(* IEC 61131-3 sources: Wago_IOWalkTest/Device/Application/FBs, 4 files *)

(* ---- FB_AITest.st ---- *)
FUNCTION_BLOCK FB_AITest
VAR_INPUT
    bStart          : BOOL;
    bStop           : BOOL;
    bSkip           : BOOL;
    bContinue       : BOOL;        // Operator presses between passes
    bStartWireBreak : BOOL;        // Start optional wire break pass
    bRetestOnly     : BOOL;
END_VAR
VAR_OUTPUT
    eState          : E_TestState;
    nCurrentChannel : INT;
    nCurrentPass    : INT;         // 1=4mA, 2=12mA, 3=20mA, 4=wirebreak
    nTotalChannels  : INT := GVL_IOWalkTest.C_NUM_AI;
    aReadings       : ARRAY[0..31, 1..3] OF INT;
    aResults        : ARRAY[0..31, 1..4] OF E_TestResult;  // 4th = wire break
    sCurrentAddress : STRING(15);
    sCurrentTag     : STRING(40);
    sCurrentDesc    : STRING(80);
    sCurrentUnit    : STRING(15);
    nCurrentRaw     : INT;
    nExpectedRaw    : INT;
    rCurrentScaled  : REAL;
    rExpectedScaled : REAL;
    rErrorPct       : REAL;
    rMaxErrorPct    : REAL;
    bSignalDetected : BOOL;
    bSettling       : BOOL;
    nPassed         : INT;
    nFailed         : INT;
    bAlmTimeout     : BOOL;
    bWireBreakDone  : BOOL;
END_VAR
VAR
    fbSettle        : TON;
    fbTimeout       : TON;
    aAI_Channels    : ARRAY[0..31] OF ST_AIChannel;
    bStartPrev      : BOOL;
    bSkipPrev       : BOOL;
    bContinuePrev   : BOOL;
    bWireBreakPrev  : BOOL;
    i               : INT;
    nRaw            : INT;
    bInWindow       : BOOL;
    rScaledActual   : REAL;
    rScaledExpected : REAL;
    rSpan           : REAL;
    rErr            : REAL;
END_VAR

// One-shot start
IF bStart AND NOT bStartPrev THEN
    IF eState = E_TestState.IDLE OR eState = E_TestState.COMPLETE OR eState = E_TestState.ABORTED THEN
        eState := E_TestState.RUNNING;
        nCurrentChannel := 0;
        nCurrentPass := 1;
        nPassed := 0;
        nFailed := 0;
        rMaxErrorPct := 0.0;
        bAlmTimeout := FALSE;
        bWireBreakDone := FALSE;
        fbSettle(IN := FALSE);
        fbTimeout(IN := FALSE);

        IF NOT bRetestOnly THEN
            FOR i := 0 TO 31 DO
                aResults[i, 1] := E_TestResult.UNTESTED;
                aResults[i, 2] := E_TestResult.UNTESTED;
                aResults[i, 3] := E_TestResult.UNTESTED;
                aResults[i, 4] := E_TestResult.UNTESTED;
            END_FOR
        END_IF
    END_IF
END_IF
bStartPrev := bStart;

// Stop
IF bStop THEN
    IF eState = E_TestState.RUNNING OR eState = E_TestState.WAIT_CONTINUE THEN
        eState := E_TestState.ABORTED;
        fbSettle(IN := FALSE);
        fbTimeout(IN := FALSE);
    END_IF
END_IF

// Continue between passes (one-shot)
IF bContinue AND NOT bContinuePrev AND eState = E_TestState.WAIT_CONTINUE THEN
    eState := E_TestState.RUNNING;
    fbTimeout(IN := FALSE);
END_IF
bContinuePrev := bContinue;

// Skip channel (one-shot)
IF bSkip AND NOT bSkipPrev AND eState = E_TestState.RUNNING THEN
    aResults[nCurrentChannel, nCurrentPass] := E_TestResult.SKIPPED;
    fbSettle(IN := FALSE);
    fbTimeout(IN := FALSE);
    nCurrentChannel := nCurrentChannel + 1;

    IF nCurrentChannel >= nTotalChannels THEN
        IF nCurrentPass < 3 THEN
            eState := E_TestState.WAIT_CONTINUE;
            nCurrentChannel := 0;
            nCurrentPass := nCurrentPass + 1;
        ELSE
            eState := E_TestState.COMPLETE;
        END_IF
    END_IF
END_IF
bSkipPrev := bSkip;

// Wire break test (one-shot)
IF bStartWireBreak AND NOT bWireBreakPrev THEN
    IF eState = E_TestState.COMPLETE OR eState = E_TestState.IDLE THEN
        nCurrentPass := 4;
        bWireBreakDone := FALSE;

        FOR i := 0 TO nTotalChannels - 1 DO
            IF aAI_Channels[i].pInput <> 0 THEN
                nRaw := aAI_Channels[i].pInput^;
                IF nRaw < GVL_IOWalkTest.C_AI_WIREBREAK_MAX THEN
                    aResults[i, 4] := E_TestResult.PASSED;
                    nPassed := nPassed + 1;
                ELSE
                    aResults[i, 4] := E_TestResult.FAILED;
                    nFailed := nFailed + 1;
                END_IF
            END_IF
        END_FOR

        bWireBreakDone := TRUE;
    END_IF
END_IF
bWireBreakPrev := bStartWireBreak;

// Main test logic (passes 1-3)
IF eState = E_TestState.RUNNING AND nCurrentPass >= 1 AND nCurrentPass <= 3
   AND nCurrentChannel < nTotalChannels THEN

    // Update HMI info
    sCurrentAddress := aAI_Channels[nCurrentChannel].sAddress;
    sCurrentTag     := aAI_Channels[nCurrentChannel].sTag;
    sCurrentDesc    := aAI_Channels[nCurrentChannel].sDescription;
    sCurrentUnit    := aAI_Channels[nCurrentChannel].sUnit;
    nExpectedRaw    := GVL_IOWalkTest.C_AI_EXPECTED_RAW[nCurrentPass];

    // Read current raw value
    IF aAI_Channels[nCurrentChannel].pInput <> 0 THEN
        nCurrentRaw := aAI_Channels[nCurrentChannel].pInput^;
    END_IF

    // Scale for display
    rSpan := aAI_Channels[nCurrentChannel].rRangeHigh - aAI_Channels[nCurrentChannel].rRangeLow;
    IF rSpan > 0.0 THEN
        rCurrentScaled  := aAI_Channels[nCurrentChannel].rRangeLow
                           + (INT_TO_REAL(nCurrentRaw) / 32767.0) * rSpan;
        rExpectedScaled := aAI_Channels[nCurrentChannel].rRangeLow
                           + (INT_TO_REAL(nExpectedRaw) / 32767.0) * rSpan;
    END_IF

    // Channel timeout
    fbTimeout(IN := TRUE, PT := GVL_IOWalkTest.C_AI_TIMEOUT);

    // Check if signal is within expected window
    bInWindow := ABS(nCurrentRaw - nExpectedRaw) < GVL_IOWalkTest.C_AI_RAW_TOLERANCE;
    bSignalDetected := bInWindow;

    IF bInWindow THEN
        // Settle timer
        fbSettle(IN := TRUE, PT := GVL_IOWalkTest.C_AI_SETTLE_TIME);
        bSettling := TRUE;

        IF fbSettle.Q THEN
            // Record reading
            aReadings[nCurrentChannel, nCurrentPass] := nCurrentRaw;

            // Evaluate pass/fail
            rScaledActual   := aAI_Channels[nCurrentChannel].rRangeLow
                               + (INT_TO_REAL(nCurrentRaw) / 32767.0) * rSpan;
            rScaledExpected := aAI_Channels[nCurrentChannel].rRangeLow
                               + (INT_TO_REAL(nExpectedRaw) / 32767.0) * rSpan;

            IF rSpan > 0.0 THEN
                rErr := ABS(rScaledActual - rScaledExpected) / rSpan * 100.0;
            ELSE
                rErr := 0.0;
            END_IF

            rErrorPct := rErr;
            IF rErr > rMaxErrorPct THEN
                rMaxErrorPct := rErr;
            END_IF

            IF rErr < GVL_IOWalkTest.C_AI_ERROR_PCT_MAX THEN
                aResults[nCurrentChannel, nCurrentPass] := E_TestResult.PASSED;
                nPassed := nPassed + 1;
            ELSE
                aResults[nCurrentChannel, nCurrentPass] := E_TestResult.FAILED;
                nFailed := nFailed + 1;
            END_IF

            // Advance
            fbSettle(IN := FALSE);
            fbTimeout(IN := FALSE);
            bSettling := FALSE;
            nCurrentChannel := nCurrentChannel + 1;

            IF nCurrentChannel >= nTotalChannels THEN
                IF nCurrentPass < 3 THEN
                    eState := E_TestState.WAIT_CONTINUE;
                    nCurrentChannel := 0;
                    nCurrentPass := nCurrentPass + 1;
                ELSE
                    eState := E_TestState.COMPLETE;
                END_IF
            END_IF
        END_IF
    ELSE
        fbSettle(IN := FALSE);
        bSettling := FALSE;
    END_IF

    // Timeout
    IF fbTimeout.Q THEN
        aResults[nCurrentChannel, nCurrentPass] := E_TestResult.FAILED;
        nFailed := nFailed + 1;
        bAlmTimeout := TRUE;
        fbSettle(IN := FALSE);
        fbTimeout(IN := FALSE);
        bSettling := FALSE;
        nCurrentChannel := nCurrentChannel + 1;

        IF nCurrentChannel >= nTotalChannels THEN
            IF nCurrentPass < 3 THEN
                eState := E_TestState.WAIT_CONTINUE;
                nCurrentChannel := 0;
                nCurrentPass := nCurrentPass + 1;
            ELSE
                eState := E_TestState.COMPLETE;
            END_IF
        END_IF
    END_IF
END_IF

(* ---- FB_AOTest.st ---- *)
FUNCTION_BLOCK FB_AOTest
VAR_INPUT
    bStart      : BOOL;
    bStop       : BOOL;
    bSkip       : BOOL;
    bPause      : BOOL;
    bMarkFail   : BOOL;
    bRetestOnly : BOOL;
END_VAR
VAR_OUTPUT
    eState          : E_TestState;
    nCurrentChannel : INT;
    nTotalChannels  : INT := GVL_IOWalkTest.C_NUM_AO;
    aResults        : ARRAY[0..11] OF E_TestResult;
    ePhase          : E_AOPhase;
    sCurrentAddress : STRING(15);
    sCurrentTag     : STRING(40);
    sCurrentDesc    : STRING(80);
    sNextAddress    : STRING(15);
    sNextTag        : STRING(40);
    rCurrentOutput_mA : REAL;
    rRampProgress   : REAL;       // 0.0 to 1.0
    nPassed         : INT;
    nFailed         : INT;
    nSkipped        : INT;
END_VAR
VAR
    fbRampTimer     : TON;
    aAO_Channels    : ARRAY[0..11] OF ST_AOChannel;
    bStartPrev      : BOOL;
    bSkipPrev       : BOOL;
    bMarkFailPrev   : BOOL;
    bChannelMarkedFail : BOOL;
    nOutputRaw      : INT;
    rProgress       : REAL;
    tCurrentPT      : TIME;
    i               : INT;
END_VAR

// One-shot start
IF bStart AND NOT bStartPrev THEN
    IF eState = E_TestState.IDLE OR eState = E_TestState.COMPLETE OR eState = E_TestState.ABORTED THEN
        eState := E_TestState.RUNNING;
        nCurrentChannel := 0;
        ePhase := E_AOPhase.RAMP_UP;
        nPassed := 0;
        nFailed := 0;
        nSkipped := 0;
        bChannelMarkedFail := FALSE;
        fbRampTimer(IN := FALSE);

        IF NOT bRetestOnly THEN
            FOR i := 0 TO 11 DO
                aResults[i] := E_TestResult.UNTESTED;
            END_FOR
        END_IF

        // Zero all outputs
        FOR i := 0 TO 11 DO
            IF aAO_Channels[i].pOutput <> 0 THEN
                aAO_Channels[i].pOutput^ := 0;
            END_IF
        END_FOR

        IF bRetestOnly THEN
            WHILE nCurrentChannel < nTotalChannels
                  AND aResults[nCurrentChannel] = E_TestResult.PASSED DO
                nCurrentChannel := nCurrentChannel + 1;
            END_WHILE
        END_IF
    END_IF
END_IF
bStartPrev := bStart;

// Stop / All Off
IF bStop THEN
    FOR i := 0 TO 11 DO
        IF aAO_Channels[i].pOutput <> 0 THEN
            aAO_Channels[i].pOutput^ := 0;
        END_IF
    END_FOR
    IF eState = E_TestState.RUNNING OR eState = E_TestState.PAUSED THEN
        eState := E_TestState.ABORTED;
        fbRampTimer(IN := FALSE);
    END_IF
END_IF

// Pause toggle
IF bPause AND eState = E_TestState.RUNNING THEN
    eState := E_TestState.PAUSED;
ELSIF bPause AND eState = E_TestState.PAUSED THEN
    eState := E_TestState.RUNNING;
END_IF

// Skip (one-shot)
IF bSkip AND NOT bSkipPrev AND eState = E_TestState.RUNNING THEN
    IF aAO_Channels[nCurrentChannel].pOutput <> 0 THEN
        aAO_Channels[nCurrentChannel].pOutput^ := 0;
    END_IF
    aResults[nCurrentChannel] := E_TestResult.SKIPPED;
    nSkipped := nSkipped + 1;
    bChannelMarkedFail := FALSE;
    fbRampTimer(IN := FALSE);
    ePhase := E_AOPhase.RAMP_UP;
    nCurrentChannel := nCurrentChannel + 1;

    IF bRetestOnly THEN
        WHILE nCurrentChannel < nTotalChannels
              AND aResults[nCurrentChannel] = E_TestResult.PASSED DO
            nCurrentChannel := nCurrentChannel + 1;
        END_WHILE
    END_IF

    IF nCurrentChannel >= nTotalChannels THEN
        eState := E_TestState.COMPLETE;
    END_IF
END_IF
bSkipPrev := bSkip;

// Mark fail (one-shot)
IF bMarkFail AND NOT bMarkFailPrev AND eState = E_TestState.RUNNING THEN
    bChannelMarkedFail := TRUE;
END_IF
bMarkFailPrev := bMarkFail;

// Main ramp logic
IF eState = E_TestState.RUNNING AND nCurrentChannel < nTotalChannels THEN
    // HMI info
    sCurrentAddress := aAO_Channels[nCurrentChannel].sAddress;
    sCurrentTag     := aAO_Channels[nCurrentChannel].sTag;
    sCurrentDesc    := aAO_Channels[nCurrentChannel].sDescription;

    IF nCurrentChannel + 1 < nTotalChannels THEN
        sNextAddress := aAO_Channels[nCurrentChannel + 1].sAddress;
        sNextTag     := aAO_Channels[nCurrentChannel + 1].sTag;
    ELSE
        sNextAddress := '';
        sNextTag     := '(last channel)';
    END_IF

    // Select timer preset based on phase
    CASE ePhase OF
        E_AOPhase.RAMP_UP, E_AOPhase.RAMP_DOWN:
            tCurrentPT := GVL_IOWalkTest.C_AO_RAMP_TIME;
        E_AOPhase.PAUSE:
            tCurrentPT := GVL_IOWalkTest.C_AO_PAUSE_TIME;
    END_CASE

    fbRampTimer(IN := TRUE, PT := tCurrentPT);
    rProgress := TIME_TO_REAL(fbRampTimer.ET) / TIME_TO_REAL(tCurrentPT);
    IF rProgress > 1.0 THEN rProgress := 1.0; END_IF
    rRampProgress := rProgress;

    CASE ePhase OF
    E_AOPhase.RAMP_UP:
        // 4mA -> 20mA (raw 0 -> 32767)
        nOutputRaw := REAL_TO_INT(rProgress * 32767.0);
        IF aAO_Channels[nCurrentChannel].pOutput <> 0 THEN
            aAO_Channels[nCurrentChannel].pOutput^ := nOutputRaw;
        END_IF
        rCurrentOutput_mA := 4.0 + (rProgress * 16.0);

        IF fbRampTimer.Q THEN
            fbRampTimer(IN := FALSE);
            ePhase := E_AOPhase.RAMP_DOWN;
        END_IF

    E_AOPhase.RAMP_DOWN:
        // 20mA -> 4mA (raw 32767 -> 0)
        nOutputRaw := REAL_TO_INT((1.0 - rProgress) * 32767.0);
        IF aAO_Channels[nCurrentChannel].pOutput <> 0 THEN
            aAO_Channels[nCurrentChannel].pOutput^ := nOutputRaw;
        END_IF
        rCurrentOutput_mA := 4.0 + ((1.0 - rProgress) * 16.0);

        IF fbRampTimer.Q THEN
            IF aAO_Channels[nCurrentChannel].pOutput <> 0 THEN
                aAO_Channels[nCurrentChannel].pOutput^ := 0;
            END_IF
            fbRampTimer(IN := FALSE);
            ePhase := E_AOPhase.PAUSE;
        END_IF

    E_AOPhase.PAUSE:
        // Pause between channels
        IF aAO_Channels[nCurrentChannel].pOutput <> 0 THEN
            aAO_Channels[nCurrentChannel].pOutput^ := 0;
        END_IF
        rCurrentOutput_mA := 4.0;

        IF fbRampTimer.Q THEN
            // Record result
            IF bChannelMarkedFail THEN
                aResults[nCurrentChannel] := E_TestResult.FAILED;
                nFailed := nFailed + 1;
            ELSE
                aResults[nCurrentChannel] := E_TestResult.PASSED;
                nPassed := nPassed + 1;
            END_IF

            bChannelMarkedFail := FALSE;
            fbRampTimer(IN := FALSE);
            ePhase := E_AOPhase.RAMP_UP;
            nCurrentChannel := nCurrentChannel + 1;

            IF bRetestOnly THEN
                WHILE nCurrentChannel < nTotalChannels
                      AND aResults[nCurrentChannel] = E_TestResult.PASSED DO
                    nCurrentChannel := nCurrentChannel + 1;
                END_WHILE
            END_IF

            IF nCurrentChannel >= nTotalChannels THEN
                FOR i := 0 TO 11 DO
                    IF aAO_Channels[i].pOutput <> 0 THEN
                        aAO_Channels[i].pOutput^ := 0;
                    END_IF
                END_FOR
                eState := E_TestState.COMPLETE;
            END_IF
        END_IF
    END_CASE
END_IF

(* ---- FB_DITest.st ---- *)
FUNCTION_BLOCK FB_DITest
VAR_INPUT
    bStart          : BOOL;
    bStop           : BOOL;
    bSkip           : BOOL;
    bRetestOnly     : BOOL;     // Only retest channels that previously failed
END_VAR
VAR_OUTPUT
    eState          : E_TestState;
    nCurrentChannel : INT;
    nTotalChannels  : INT := GVL_IOWalkTest.C_NUM_DI;
    aResults        : ARRAY[0..71] OF E_TestResult;
    bWaitingForRise : BOOL;
    bWaitingForFall : BOOL;
    sCurrentAddress : STRING(15);
    sCurrentTag     : STRING(40);
    sCurrentDesc    : STRING(80);
    eCurrentContact : E_ContactType;
    nPassed         : INT;
    nFailed         : INT;
    nSkipped        : INT;
    bAlmTimeout     : BOOL;
    bAlmWrongChan   : BOOL;
    nWrongChanIdx   : INT;
END_VAR
VAR
    fbTimeout       : TON;
    aDI_Prev        : ARRAY[0..71] OF BOOL;
    aDI_Channels    : ARRAY[0..71] OF ST_DIChannel;
    bInitDone       : BOOL;
    bStartPrev      : BOOL;
    bSkipPrev       : BOOL;
    i               : INT;
    bCurrentState   : BOOL;
    bPrevState      : BOOL;
    bExpectRise     : BOOL;     // TRUE = waiting for active edge
    bExpectFall     : BOOL;     // TRUE = waiting for release edge
END_VAR

// One-shot start detection
IF bStart AND NOT bStartPrev THEN
    IF eState = E_TestState.IDLE OR eState = E_TestState.COMPLETE OR eState = E_TestState.ABORTED THEN
        eState := E_TestState.RUNNING;
        nCurrentChannel := 0;
        bAlmTimeout := FALSE;
        bAlmWrongChan := FALSE;
        nPassed := 0;
        nFailed := 0;
        nSkipped := 0;
        fbTimeout(IN := FALSE);

        IF NOT bRetestOnly THEN
            FOR i := 0 TO 71 DO
                aResults[i] := E_TestResult.UNTESTED;
            END_FOR
        END_IF

        // Skip to first untested/failed channel if retest mode
        IF bRetestOnly THEN
            WHILE nCurrentChannel < nTotalChannels
                  AND aResults[nCurrentChannel] = E_TestResult.PASSED DO
                nCurrentChannel := nCurrentChannel + 1;
            END_WHILE
        END_IF

        // Determine initial edge expectations
        IF nCurrentChannel < nTotalChannels THEN
            IF aDI_Channels[nCurrentChannel].eContactType = E_ContactType.NC THEN
                bExpectRise := FALSE;
                bExpectFall := TRUE;    // NC: wait for fall first
            ELSE
                bExpectRise := TRUE;
                bExpectFall := FALSE;   // NO: wait for rise first
            END_IF
        END_IF
    END_IF
END_IF
bStartPrev := bStart;

// Stop
IF bStop THEN
    IF eState = E_TestState.RUNNING THEN
        eState := E_TestState.ABORTED;
        fbTimeout(IN := FALSE);
    END_IF
END_IF

// Skip channel (one-shot)
IF bSkip AND NOT bSkipPrev AND eState = E_TestState.RUNNING THEN
    aResults[nCurrentChannel] := E_TestResult.SKIPPED;
    nSkipped := nSkipped + 1;
    fbTimeout(IN := FALSE);
    nCurrentChannel := nCurrentChannel + 1;

    // Skip already-passed channels in retest mode
    IF bRetestOnly THEN
        WHILE nCurrentChannel < nTotalChannels
              AND aResults[nCurrentChannel] = E_TestResult.PASSED DO
            nCurrentChannel := nCurrentChannel + 1;
        END_WHILE
    END_IF

    IF nCurrentChannel >= nTotalChannels THEN
        eState := E_TestState.COMPLETE;
    END_IF
END_IF
bSkipPrev := bSkip;

// Main test logic
IF eState = E_TestState.RUNNING AND nCurrentChannel < nTotalChannels THEN
    // Update HMI display info
    sCurrentAddress := aDI_Channels[nCurrentChannel].sAddress;
    sCurrentTag     := aDI_Channels[nCurrentChannel].sTag;
    sCurrentDesc    := aDI_Channels[nCurrentChannel].sDescription;
    eCurrentContact := aDI_Channels[nCurrentChannel].eContactType;

    // Read current channel state via pointer
    IF aDI_Channels[nCurrentChannel].pInput <> 0 THEN
        bCurrentState := aDI_Channels[nCurrentChannel].pInput^;
    END_IF
    bPrevState := aDI_Prev[nCurrentChannel];

    // Channel timeout
    fbTimeout(IN := TRUE, PT := GVL_IOWalkTest.C_DI_TIMEOUT);

    // Edge detection based on contact type
    // NO contacts: rise then fall
    // NC contacts: fall then rise (inverted)
    IF bExpectRise AND bCurrentState AND NOT bPrevState THEN
        // Rising edge detected
        bExpectRise := FALSE;
        bExpectFall := TRUE;
        fbTimeout(IN := FALSE);
        fbTimeout(IN := TRUE, PT := GVL_IOWalkTest.C_DI_TIMEOUT);
    END_IF

    IF bExpectFall AND NOT bCurrentState AND bPrevState THEN
        // Falling edge detected - channel PASS
        aResults[nCurrentChannel] := E_TestResult.PASSED;
        nPassed := nPassed + 1;
        fbTimeout(IN := FALSE);

        // Advance
        nCurrentChannel := nCurrentChannel + 1;

        // Skip already-passed in retest mode
        IF bRetestOnly THEN
            WHILE nCurrentChannel < nTotalChannels
                  AND aResults[nCurrentChannel] = E_TestResult.PASSED DO
                nCurrentChannel := nCurrentChannel + 1;
            END_WHILE
        END_IF

        IF nCurrentChannel >= nTotalChannels THEN
            eState := E_TestState.COMPLETE;
        ELSE
            // Set up edge expectations for next channel
            IF aDI_Channels[nCurrentChannel].eContactType = E_ContactType.NC THEN
                bExpectRise := FALSE;
                bExpectFall := TRUE;
            ELSE
                bExpectRise := TRUE;
                bExpectFall := FALSE;
            END_IF
            fbTimeout(IN := TRUE, PT := GVL_IOWalkTest.C_DI_TIMEOUT);
        END_IF
    END_IF

    // Check for out-of-order channel activation
    FOR i := 0 TO nTotalChannels - 1 DO
        IF i <> nCurrentChannel AND aDI_Channels[i].pInput <> 0 THEN
            IF aDI_Channels[i].pInput^ AND NOT aDI_Prev[i] THEN
                bAlmWrongChan := TRUE;
                nWrongChanIdx := i;
            END_IF
        END_IF
    END_FOR

    // Timeout handling
    IF fbTimeout.Q THEN
        aResults[nCurrentChannel] := E_TestResult.FAILED;
        nFailed := nFailed + 1;
        bAlmTimeout := TRUE;
        fbTimeout(IN := FALSE);

        nCurrentChannel := nCurrentChannel + 1;
        IF bRetestOnly THEN
            WHILE nCurrentChannel < nTotalChannels
                  AND aResults[nCurrentChannel] = E_TestResult.PASSED DO
                nCurrentChannel := nCurrentChannel + 1;
            END_WHILE
        END_IF

        IF nCurrentChannel >= nTotalChannels THEN
            eState := E_TestState.COMPLETE;
        ELSE
            IF aDI_Channels[nCurrentChannel].eContactType = E_ContactType.NC THEN
                bExpectRise := FALSE;
                bExpectFall := TRUE;
            ELSE
                bExpectRise := TRUE;
                bExpectFall := FALSE;
            END_IF
            fbTimeout(IN := TRUE, PT := GVL_IOWalkTest.C_DI_TIMEOUT);
        END_IF
    END_IF

    // Store previous states for all channels
    FOR i := 0 TO nTotalChannels - 1 DO
        IF aDI_Channels[i].pInput <> 0 THEN
            aDI_Prev[i] := aDI_Channels[i].pInput^;
        END_IF
    END_FOR
END_IF

(* ---- FB_DOTest.st ---- *)
FUNCTION_BLOCK FB_DOTest
VAR_INPUT
    bStart      : BOOL;
    bStop       : BOOL;
    bSkip       : BOOL;
    bPause      : BOOL;
    bMarkFail   : BOOL;
    bRetestOnly : BOOL;
END_VAR
VAR_OUTPUT
    eState          : E_TestState;
    nCurrentChannel : INT;
    nTotalChannels  : INT := GVL_IOWalkTest.C_NUM_DO;
    aResults        : ARRAY[0..55] OF E_TestResult;
    sCurrentAddress : STRING(15);
    sCurrentTag     : STRING(40);
    sCurrentDesc    : STRING(80);
    sCurrentNote    : STRING(120);
    sNextAddress    : STRING(15);
    sNextTag        : STRING(40);
    rSecondsRemain  : REAL;
    nPassed         : INT;
    nFailed         : INT;
    nSkipped        : INT;
END_VAR
VAR
    fbDwell         : TON;
    aDO_Channels    : ARRAY[0..55] OF ST_DOChannel;
    bStartPrev      : BOOL;
    bSkipPrev       : BOOL;
    bMarkFailPrev   : BOOL;
    bChannelMarkedFail : BOOL;
    i               : INT;
END_VAR

// One-shot start
IF bStart AND NOT bStartPrev THEN
    IF eState = E_TestState.IDLE OR eState = E_TestState.COMPLETE OR eState = E_TestState.ABORTED THEN
        eState := E_TestState.RUNNING;
        nCurrentChannel := 0;
        nPassed := 0;
        nFailed := 0;
        nSkipped := 0;
        bChannelMarkedFail := FALSE;
        fbDwell(IN := FALSE);

        IF NOT bRetestOnly THEN
            FOR i := 0 TO 55 DO
                aResults[i] := E_TestResult.UNTESTED;
            END_FOR
        END_IF

        // De-energize all outputs
        FOR i := 0 TO 55 DO
            IF aDO_Channels[i].pOutput <> 0 THEN
                aDO_Channels[i].pOutput^ := FALSE;
            END_IF
        END_FOR

        // Skip passed channels in retest mode
        IF bRetestOnly THEN
            WHILE nCurrentChannel < nTotalChannels
                  AND aResults[nCurrentChannel] = E_TestResult.PASSED DO
                nCurrentChannel := nCurrentChannel + 1;
            END_WHILE
        END_IF
    END_IF
END_IF
bStartPrev := bStart;

// Stop / All Off
IF bStop THEN
    FOR i := 0 TO 55 DO
        IF aDO_Channels[i].pOutput <> 0 THEN
            aDO_Channels[i].pOutput^ := FALSE;
        END_IF
    END_FOR
    IF eState = E_TestState.RUNNING OR eState = E_TestState.PAUSED THEN
        eState := E_TestState.ABORTED;
        fbDwell(IN := FALSE);
    END_IF
END_IF

// Pause toggle
IF bPause AND eState = E_TestState.RUNNING THEN
    eState := E_TestState.PAUSED;
ELSIF bPause AND eState = E_TestState.PAUSED THEN
    eState := E_TestState.RUNNING;
END_IF

// Skip channel (one-shot)
IF bSkip AND NOT bSkipPrev AND (eState = E_TestState.RUNNING OR eState = E_TestState.PAUSED) THEN
    IF aDO_Channels[nCurrentChannel].pOutput <> 0 THEN
        aDO_Channels[nCurrentChannel].pOutput^ := FALSE;
    END_IF
    aResults[nCurrentChannel] := E_TestResult.SKIPPED;
    nSkipped := nSkipped + 1;
    fbDwell(IN := FALSE);
    bChannelMarkedFail := FALSE;
    nCurrentChannel := nCurrentChannel + 1;

    IF bRetestOnly THEN
        WHILE nCurrentChannel < nTotalChannels
              AND aResults[nCurrentChannel] = E_TestResult.PASSED DO
            nCurrentChannel := nCurrentChannel + 1;
        END_WHILE
    END_IF

    IF nCurrentChannel >= nTotalChannels THEN
        eState := E_TestState.COMPLETE;
    END_IF
END_IF
bSkipPrev := bSkip;

// Mark fail (one-shot)
IF bMarkFail AND NOT bMarkFailPrev AND eState = E_TestState.RUNNING THEN
    bChannelMarkedFail := TRUE;
END_IF
bMarkFailPrev := bMarkFail;

// Main sequencing logic
IF eState = E_TestState.RUNNING AND nCurrentChannel < nTotalChannels THEN
    // Update HMI info
    sCurrentAddress := aDO_Channels[nCurrentChannel].sAddress;
    sCurrentTag     := aDO_Channels[nCurrentChannel].sTag;
    sCurrentDesc    := aDO_Channels[nCurrentChannel].sDescription;
    sCurrentNote    := aDO_Channels[nCurrentChannel].sNote;

    IF nCurrentChannel + 1 < nTotalChannels THEN
        sNextAddress := aDO_Channels[nCurrentChannel + 1].sAddress;
        sNextTag     := aDO_Channels[nCurrentChannel + 1].sTag;
    ELSE
        sNextAddress := '';
        sNextTag     := '(last channel)';
    END_IF

    // Energize current channel
    IF aDO_Channels[nCurrentChannel].pOutput <> 0 THEN
        aDO_Channels[nCurrentChannel].pOutput^ := TRUE;
    END_IF

    // Dwell timer
    fbDwell(IN := TRUE, PT := GVL_IOWalkTest.C_DO_DWELL_TIME);
    rSecondsRemain := TIME_TO_REAL(GVL_IOWalkTest.C_DO_DWELL_TIME - fbDwell.ET) / 1000.0;

    IF fbDwell.Q THEN
        // De-energize
        IF aDO_Channels[nCurrentChannel].pOutput <> 0 THEN
            aDO_Channels[nCurrentChannel].pOutput^ := FALSE;
        END_IF

        // Record result
        IF bChannelMarkedFail THEN
            aResults[nCurrentChannel] := E_TestResult.FAILED;
            nFailed := nFailed + 1;
        ELSE
            aResults[nCurrentChannel] := E_TestResult.PASSED;
            nPassed := nPassed + 1;
        END_IF

        bChannelMarkedFail := FALSE;
        fbDwell(IN := FALSE);
        nCurrentChannel := nCurrentChannel + 1;

        IF bRetestOnly THEN
            WHILE nCurrentChannel < nTotalChannels
                  AND aResults[nCurrentChannel] = E_TestResult.PASSED DO
                nCurrentChannel := nCurrentChannel + 1;
            END_WHILE
        END_IF

        IF nCurrentChannel >= nTotalChannels THEN
            // De-energize all
            FOR i := 0 TO 55 DO
                IF aDO_Channels[i].pOutput <> 0 THEN
                    aDO_Channels[i].pOutput^ := FALSE;
                END_IF
            END_FOR
            eState := E_TestState.COMPLETE;
        END_IF
    END_IF
END_IF
